// TIA Portal V18 export
// export: Created 2026-06-14T13:43:50.166899Z, ExportSetting WithDefaults, DisplayName Totally Integrated Automation Portal, DisplayVersion V18 Update 5, DisplayName TIA Portal Openness, DisplayVersion V18 Update 5, DisplayName TIA Portal Version Control Interface, DisplayVersion V18, DisplayName SINAMICS Startdrive Advanced, DisplayVersion V18 SP2 Update 1, DisplayName SINAMICS Startdrive G110M, G120, G120C, G120D, G120P, G115D, DisplayVersion V18 SP2 Update 1, DisplayName SINAMICS Startdrive G130, G150, S120, S150, SINAMICS MV, S210, G220, S200, DisplayVersion V18 SP2 Update 1, DisplayName STEP 7 Professional, DisplayVersion V18 Update 5, DisplayName STEP 7 Safety, DisplayVersion V18, DisplayName WinCC Advanced / Unified PC, DisplayVersion V18 Update 5
FUNCTION "TEMPLATE--v1.1--05_Output Feedback" : Void   // FC6, F_FBD
TITLE = Manage Safety Outputs
{ S7_Optimized_Access := 'TRUE' }
VERSION : 0.1
// v1.0 First Emission
// v1.1 Added 03_FDBACK_RAW reference
// stored: AutoNumber true, IsIECCheckEnabled false, UDAEnableTagReadback false
   VAR_TEMP
      DU_EX : Bool;
      ISPC_EX : Bool;
      ZONE_EX : Bool;
   END_VAR
BEGIN

REGION Network 1: !!NetworkComment$$ 1c -1i -1q
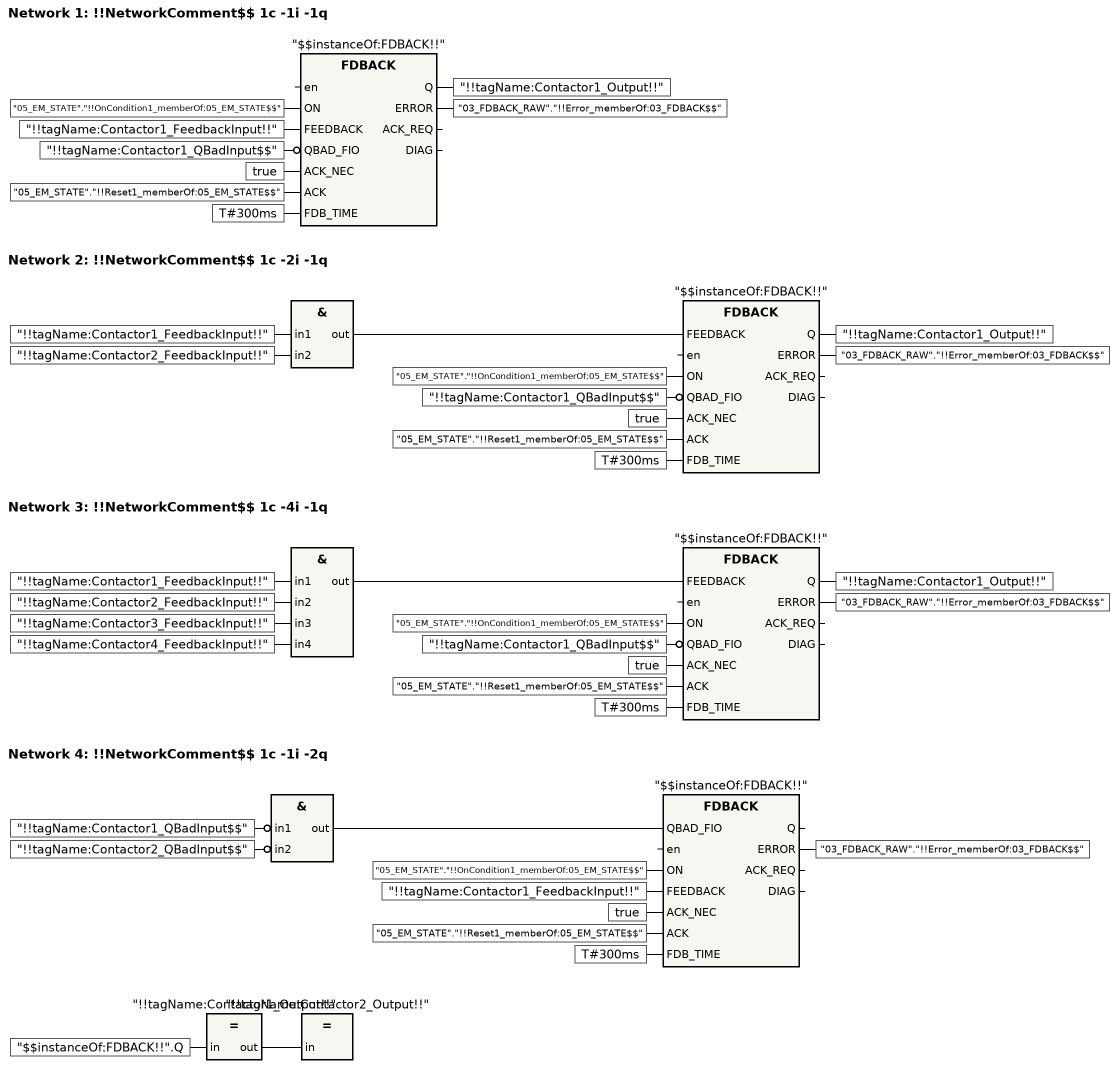
   "$$instanceOf:FDBACK!!"(ON := "05_EM_STATE"."!!OnCondition1_memberOf:05_EM_STATE$$",   // FDBACK
                           FEEDBACK := "!!tagName:Contactor1_FeedbackInput!!",
                           QBAD_FIO := NOT "!!tagName:Contactor1_QBadInput$$",
                           ACK_NEC := true,
                           ACK := "05_EM_STATE"."!!Reset1_memberOf:05_EM_STATE$$",
                           FDB_TIME := T#300ms,
                           Q => "!!tagName:Contactor1_Output!!",
                           ERROR => "03_FDBACK_RAW"."!!Error_memberOf:03_FDBACK$$");
END_REGION

REGION Network 2: !!NetworkComment$$ 1c -2i -1q
   "$$instanceOf:FDBACK!!"(FEEDBACK := "!!tagName:Contactor1_FeedbackInput!!" AND "!!tagName:Contactor2_FeedbackInput!!",   // FDBACK
                           ON := "05_EM_STATE"."!!OnCondition1_memberOf:05_EM_STATE$$",
                           QBAD_FIO := NOT "!!tagName:Contactor1_QBadInput$$",
                           ACK_NEC := true,
                           ACK := "05_EM_STATE"."!!Reset1_memberOf:05_EM_STATE$$",
                           FDB_TIME := T#300ms,
                           Q => "!!tagName:Contactor1_Output!!",
                           ERROR => "03_FDBACK_RAW"."!!Error_memberOf:03_FDBACK$$");
END_REGION

REGION Network 3: !!NetworkComment$$ 1c -4i -1q
   "$$instanceOf:FDBACK!!"(FEEDBACK := "!!tagName:Contactor1_FeedbackInput!!" AND "!!tagName:Contactor2_FeedbackInput!!" AND "!!tagName:Contactor3_FeedbackInput!!" AND "!!tagName:Contactor4_FeedbackInput!!",   // FDBACK
                           ON := "05_EM_STATE"."!!OnCondition1_memberOf:05_EM_STATE$$",
                           QBAD_FIO := NOT "!!tagName:Contactor1_QBadInput$$",
                           ACK_NEC := true,
                           ACK := "05_EM_STATE"."!!Reset1_memberOf:05_EM_STATE$$",
                           FDB_TIME := T#300ms,
                           Q => "!!tagName:Contactor1_Output!!",
                           ERROR => "03_FDBACK_RAW"."!!Error_memberOf:03_FDBACK$$");
END_REGION

REGION Network 4: !!NetworkComment$$ 1c -1i -2q
   "$$instanceOf:FDBACK!!"(QBAD_FIO := NOT "!!tagName:Contactor1_QBadInput$$" AND NOT "!!tagName:Contactor2_QBadInput$$",   // FDBACK
                           ON := "05_EM_STATE"."!!OnCondition1_memberOf:05_EM_STATE$$",
                           FEEDBACK := "!!tagName:Contactor1_FeedbackInput!!",
                           ACK_NEC := true,
                           ACK := "05_EM_STATE"."!!Reset1_memberOf:05_EM_STATE$$",
                           FDB_TIME := T#300ms,
                           ERROR => "03_FDBACK_RAW"."!!Error_memberOf:03_FDBACK$$");
   "!!tagName:Contactor1_Output!!" := "$$instanceOf:FDBACK!!".Q;
   "!!tagName:Contactor2_Output!!" := "$$instanceOf:FDBACK!!".Q;
END_REGION

REGION Network 5: !!NetworkComment$$ 1c -2i -2q
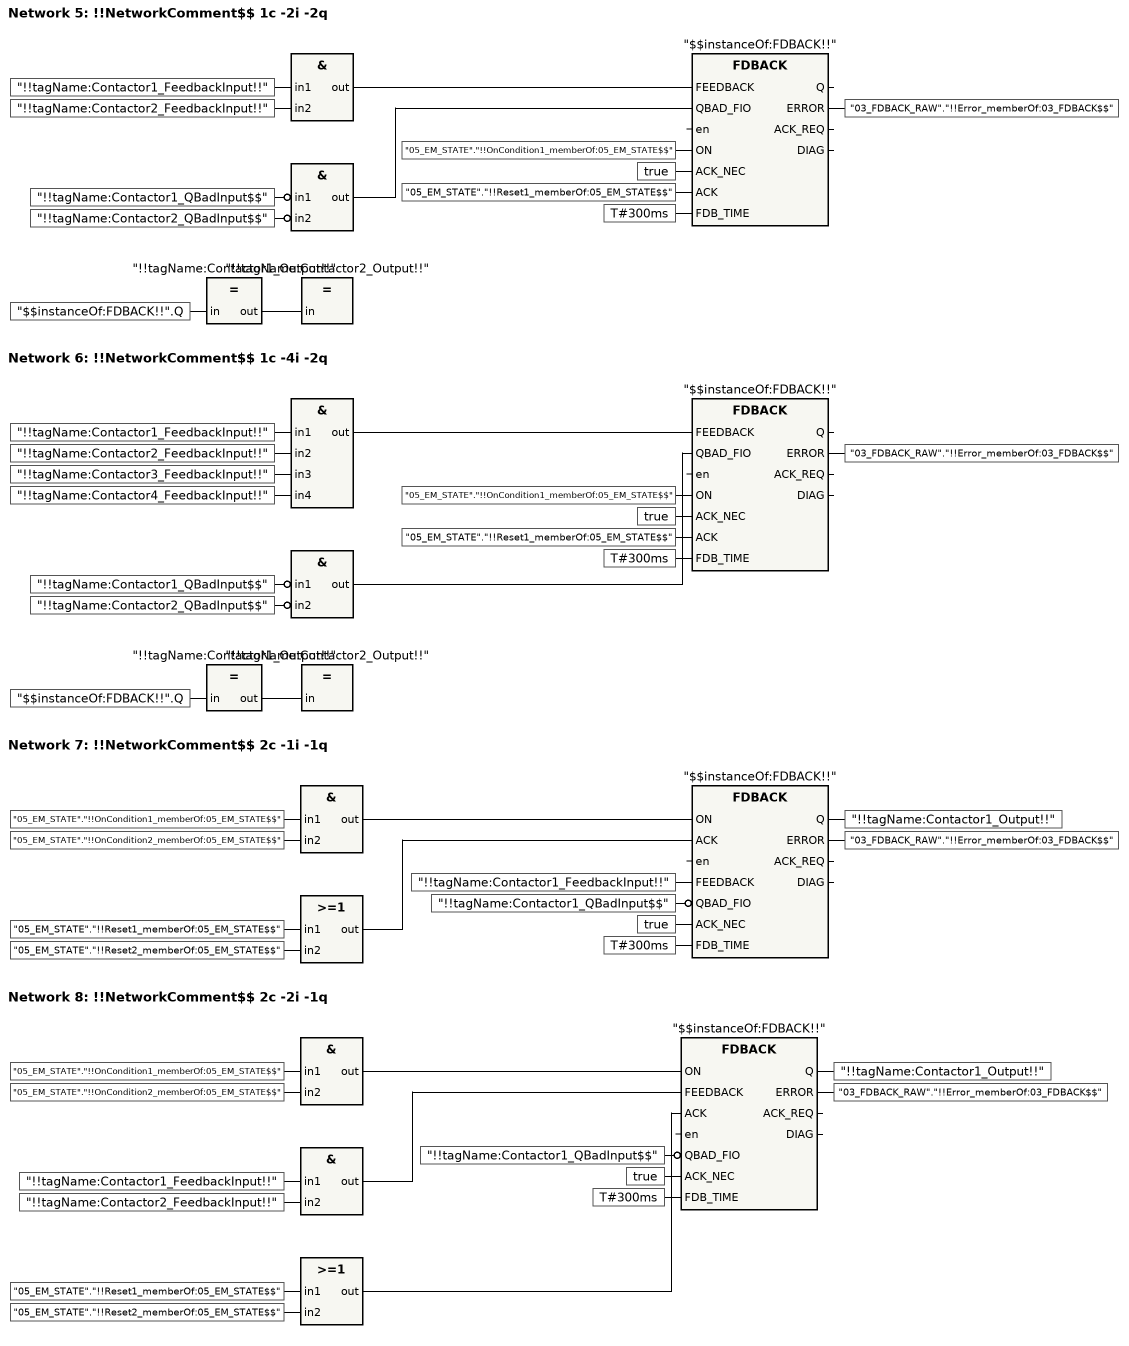
   "$$instanceOf:FDBACK!!"(FEEDBACK := "!!tagName:Contactor1_FeedbackInput!!" AND "!!tagName:Contactor2_FeedbackInput!!",   // FDBACK
                           QBAD_FIO := NOT "!!tagName:Contactor1_QBadInput$$" AND NOT "!!tagName:Contactor2_QBadInput$$",
                           ON := "05_EM_STATE"."!!OnCondition1_memberOf:05_EM_STATE$$",
                           ACK_NEC := true,
                           ACK := "05_EM_STATE"."!!Reset1_memberOf:05_EM_STATE$$",
                           FDB_TIME := T#300ms,
                           ERROR => "03_FDBACK_RAW"."!!Error_memberOf:03_FDBACK$$");
   "!!tagName:Contactor1_Output!!" := "$$instanceOf:FDBACK!!".Q;
   "!!tagName:Contactor2_Output!!" := "$$instanceOf:FDBACK!!".Q;
END_REGION

REGION Network 6: !!NetworkComment$$ 1c -4i -2q
   "$$instanceOf:FDBACK!!"(FEEDBACK := "!!tagName:Contactor1_FeedbackInput!!" AND "!!tagName:Contactor2_FeedbackInput!!" AND "!!tagName:Contactor3_FeedbackInput!!" AND "!!tagName:Contactor4_FeedbackInput!!",   // FDBACK
                           QBAD_FIO := NOT "!!tagName:Contactor1_QBadInput$$" AND NOT "!!tagName:Contactor2_QBadInput$$",
                           ON := "05_EM_STATE"."!!OnCondition1_memberOf:05_EM_STATE$$",
                           ACK_NEC := true,
                           ACK := "05_EM_STATE"."!!Reset1_memberOf:05_EM_STATE$$",
                           FDB_TIME := T#300ms,
                           ERROR => "03_FDBACK_RAW"."!!Error_memberOf:03_FDBACK$$");
   "!!tagName:Contactor1_Output!!" := "$$instanceOf:FDBACK!!".Q;
   "!!tagName:Contactor2_Output!!" := "$$instanceOf:FDBACK!!".Q;
END_REGION

REGION Network 7: !!NetworkComment$$ 2c -1i -1q
   "$$instanceOf:FDBACK!!"(ON := "05_EM_STATE"."!!OnCondition1_memberOf:05_EM_STATE$$" AND "05_EM_STATE"."!!OnCondition2_memberOf:05_EM_STATE$$",   // FDBACK
                           ACK := "05_EM_STATE"."!!Reset1_memberOf:05_EM_STATE$$" OR "05_EM_STATE"."!!Reset2_memberOf:05_EM_STATE$$",
                           FEEDBACK := "!!tagName:Contactor1_FeedbackInput!!",
                           QBAD_FIO := NOT "!!tagName:Contactor1_QBadInput$$",
                           ACK_NEC := true,
                           FDB_TIME := T#300ms,
                           Q => "!!tagName:Contactor1_Output!!",
                           ERROR => "03_FDBACK_RAW"."!!Error_memberOf:03_FDBACK$$");
END_REGION

REGION Network 8: !!NetworkComment$$ 2c -2i -1q
   "$$instanceOf:FDBACK!!"(ON := "05_EM_STATE"."!!OnCondition1_memberOf:05_EM_STATE$$" AND "05_EM_STATE"."!!OnCondition2_memberOf:05_EM_STATE$$",   // FDBACK
                           FEEDBACK := "!!tagName:Contactor1_FeedbackInput!!" AND "!!tagName:Contactor2_FeedbackInput!!",
                           ACK := "05_EM_STATE"."!!Reset1_memberOf:05_EM_STATE$$" OR "05_EM_STATE"."!!Reset2_memberOf:05_EM_STATE$$",
                           QBAD_FIO := NOT "!!tagName:Contactor1_QBadInput$$",
                           ACK_NEC := true,
                           FDB_TIME := T#300ms,
                           Q => "!!tagName:Contactor1_Output!!",
                           ERROR => "03_FDBACK_RAW"."!!Error_memberOf:03_FDBACK$$");
END_REGION

REGION Network 9: !!NetworkComment$$ 1c -4i -1q
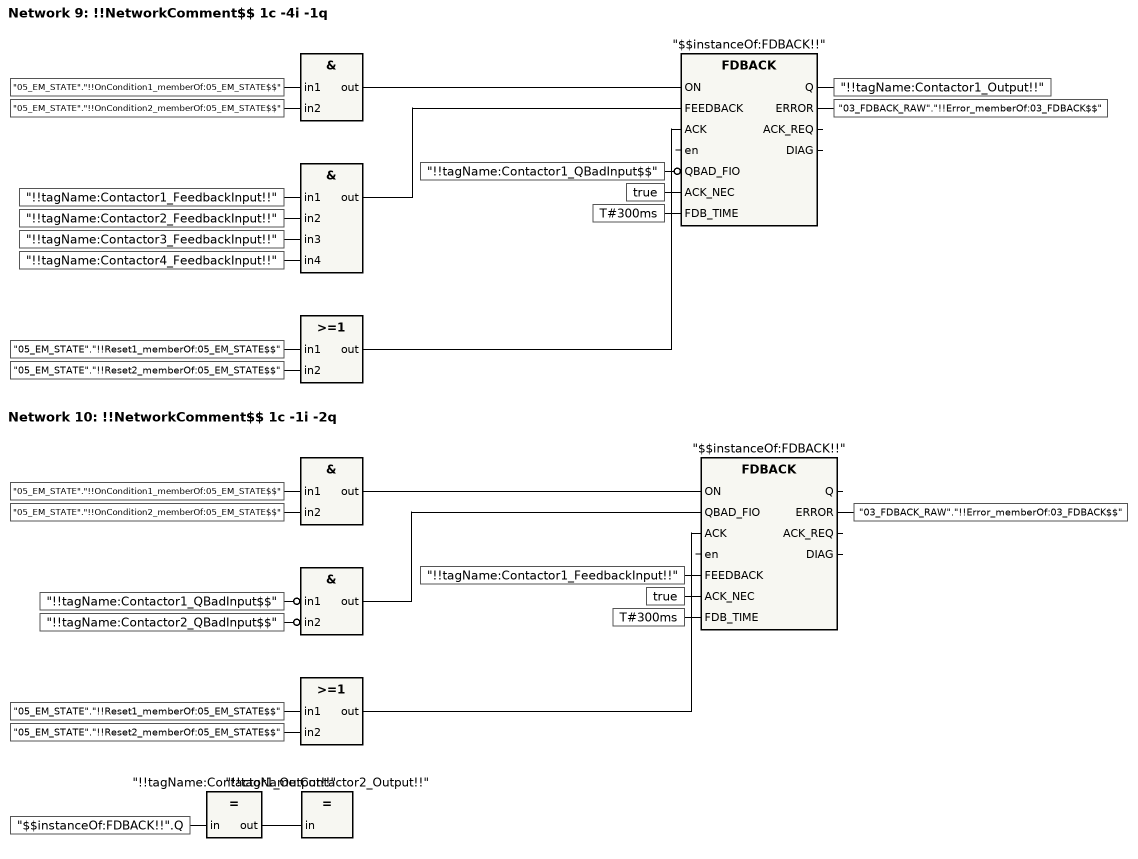
   "$$instanceOf:FDBACK!!"(ON := "05_EM_STATE"."!!OnCondition1_memberOf:05_EM_STATE$$" AND "05_EM_STATE"."!!OnCondition2_memberOf:05_EM_STATE$$",   // FDBACK
                           FEEDBACK := "!!tagName:Contactor1_FeedbackInput!!" AND "!!tagName:Contactor2_FeedbackInput!!" AND "!!tagName:Contactor3_FeedbackInput!!" AND "!!tagName:Contactor4_FeedbackInput!!",
                           ACK := "05_EM_STATE"."!!Reset1_memberOf:05_EM_STATE$$" OR "05_EM_STATE"."!!Reset2_memberOf:05_EM_STATE$$",
                           QBAD_FIO := NOT "!!tagName:Contactor1_QBadInput$$",
                           ACK_NEC := true,
                           FDB_TIME := T#300ms,
                           Q => "!!tagName:Contactor1_Output!!",
                           ERROR => "03_FDBACK_RAW"."!!Error_memberOf:03_FDBACK$$");
END_REGION

REGION Network 10: !!NetworkComment$$ 1c -1i -2q
   "$$instanceOf:FDBACK!!"(ON := "05_EM_STATE"."!!OnCondition1_memberOf:05_EM_STATE$$" AND "05_EM_STATE"."!!OnCondition2_memberOf:05_EM_STATE$$",   // FDBACK
                           QBAD_FIO := NOT "!!tagName:Contactor1_QBadInput$$" AND NOT "!!tagName:Contactor2_QBadInput$$",
                           ACK := "05_EM_STATE"."!!Reset1_memberOf:05_EM_STATE$$" OR "05_EM_STATE"."!!Reset2_memberOf:05_EM_STATE$$",
                           FEEDBACK := "!!tagName:Contactor1_FeedbackInput!!",
                           ACK_NEC := true,
                           FDB_TIME := T#300ms,
                           ERROR => "03_FDBACK_RAW"."!!Error_memberOf:03_FDBACK$$");
   "!!tagName:Contactor1_Output!!" := "$$instanceOf:FDBACK!!".Q;
   "!!tagName:Contactor2_Output!!" := "$$instanceOf:FDBACK!!".Q;
END_REGION

REGION Network 11: !!NetworkComment$$ 1c -2i -2q
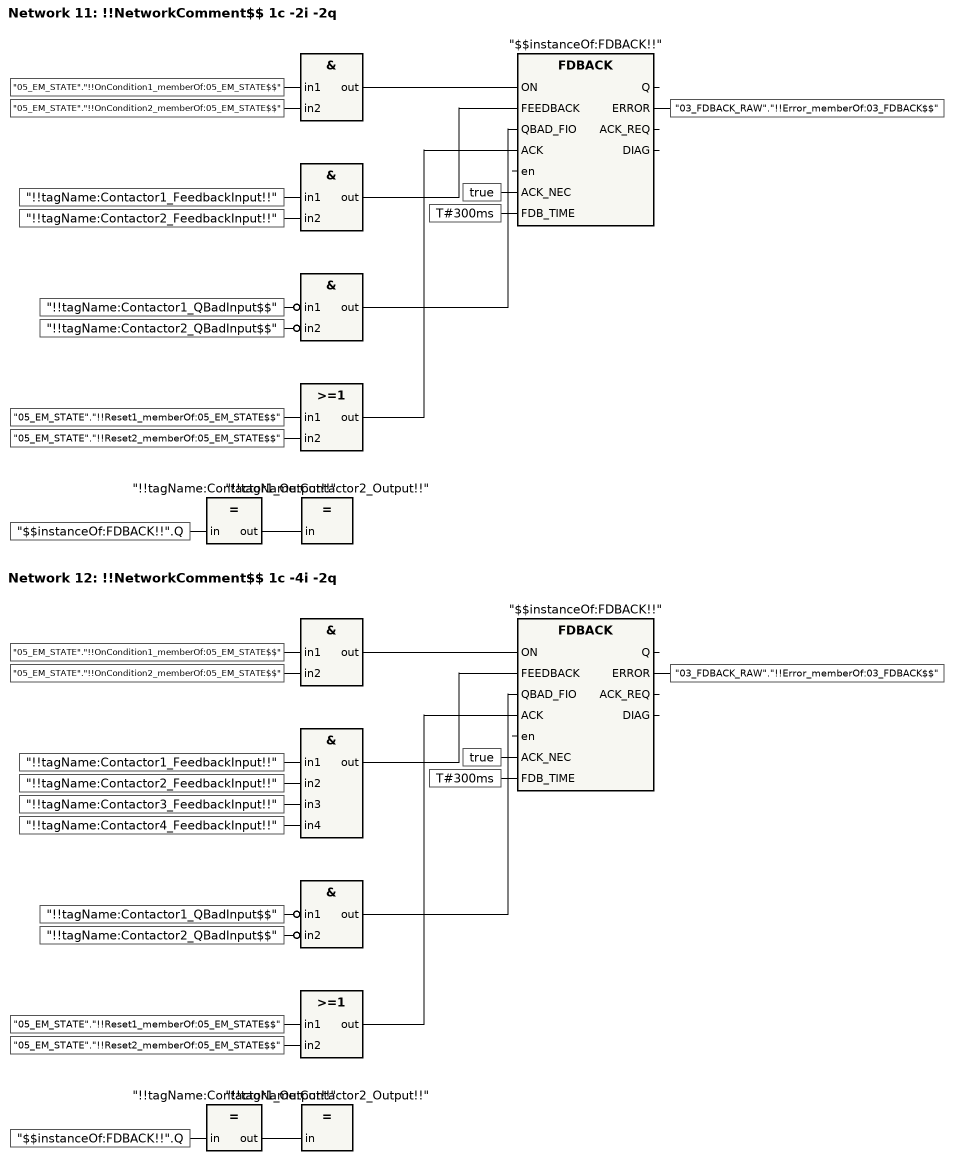
   "$$instanceOf:FDBACK!!"(ON := "05_EM_STATE"."!!OnCondition1_memberOf:05_EM_STATE$$" AND "05_EM_STATE"."!!OnCondition2_memberOf:05_EM_STATE$$",   // FDBACK
                           FEEDBACK := "!!tagName:Contactor1_FeedbackInput!!" AND "!!tagName:Contactor2_FeedbackInput!!",
                           QBAD_FIO := NOT "!!tagName:Contactor1_QBadInput$$" AND NOT "!!tagName:Contactor2_QBadInput$$",
                           ACK := "05_EM_STATE"."!!Reset1_memberOf:05_EM_STATE$$" OR "05_EM_STATE"."!!Reset2_memberOf:05_EM_STATE$$",
                           ACK_NEC := true,
                           FDB_TIME := T#300ms,
                           ERROR => "03_FDBACK_RAW"."!!Error_memberOf:03_FDBACK$$");
   "!!tagName:Contactor1_Output!!" := "$$instanceOf:FDBACK!!".Q;
   "!!tagName:Contactor2_Output!!" := "$$instanceOf:FDBACK!!".Q;
END_REGION

REGION Network 12: !!NetworkComment$$ 1c -4i -2q
   "$$instanceOf:FDBACK!!"(ON := "05_EM_STATE"."!!OnCondition1_memberOf:05_EM_STATE$$" AND "05_EM_STATE"."!!OnCondition2_memberOf:05_EM_STATE$$",   // FDBACK
                           FEEDBACK := "!!tagName:Contactor1_FeedbackInput!!" AND "!!tagName:Contactor2_FeedbackInput!!" AND "!!tagName:Contactor3_FeedbackInput!!" AND "!!tagName:Contactor4_FeedbackInput!!",
                           QBAD_FIO := NOT "!!tagName:Contactor1_QBadInput$$" AND NOT "!!tagName:Contactor2_QBadInput$$",
                           ACK := "05_EM_STATE"."!!Reset1_memberOf:05_EM_STATE$$" OR "05_EM_STATE"."!!Reset2_memberOf:05_EM_STATE$$",
                           ACK_NEC := true,
                           FDB_TIME := T#300ms,
                           ERROR => "03_FDBACK_RAW"."!!Error_memberOf:03_FDBACK$$");
   "!!tagName:Contactor1_Output!!" := "$$instanceOf:FDBACK!!".Q;
   "!!tagName:Contactor2_Output!!" := "$$instanceOf:FDBACK!!".Q;
END_REGION
END_FUNCTION
